// TIA Portal project "Digital – analógico (Ejercicio básico)" (V15.1)

(* hardware
DEVICE "S7-1200 station_2"  S7-1200 Station
   slot 0: "Rack_0"  S7-1200 Rack  Rack  V1.0
   slot 1: "PLC_2"  CPU 1214C AC/DC/Rly  6ES7 214-1BG40-0XB0  V4.1
   slot 3: "AQ 1x12BIT_1"  AQ1 signal board  6ES7 232-4HA30-0XB0  V1.0
*)

// ===== PLC "PLC_2"  CPU 1214C AC/DC/Rly =====

VAR_GLOBAL   // PLC tag table "Tabla de variables estándar"
   "etapa0" AT %M16.0 : Bool;
   "etapa1" AT %M16.1 : Bool;
   "etapa3" AT %M16.2 : Bool;
   "FC1" AT %I0.0 : Bool;
   "FC2" AT %I0.1 : Bool;
   "FC3" AT %I0.2 : Bool;
   "M" AT %I0.3 : Bool;
   "etapa2" AT %M16.3 : Bool;
   "Tag_1" AT %IW67 : Int;
   "Tag_2" AT %MD80 : Real;
   "Tag_3" AT %MD84 : Real;
   "Tag_4" AT %MD500 : DWord;
   "TAG9" AT %M500.0 : Bool;
   "Tag_5" AT %Q0.0 : Bool;
   "c100" AT %Q0.1 : Bool;
   "c10" AT %Q0.2 : Bool;
   "c-100" AT %Q0.3 : Bool;
   "Tag_6" AT %IW64 : Int;
   "Tag_7" AT %IW65 : Int;
   "Tag_8" AT %IW66 : Int;
   "Tag_9" AT %MD81 : DWord;
   "Tag_10" AT %MD82 : DWord;
   "Tag_11" AT %MD83 : DWord;
   "Tag_12" AT %IW80 : Word;
   "Tag_13" AT %IW81 : Word;
   "Tag_14" AT %MD30 : DWord;
   "Tag_15" AT %MD31 : DWord;
   "Tag_16" AT %MD32 : DWord;
   "Tag_17" AT %MD34 : Real;
   "Tag_18" AT %QW80 : Word;
END_VAR

FUNCTION "grafcet" : Void   // FC1, LAD
{ S7_Optimized_Access := 'TRUE' }
VERSION : 0.1
BEGIN

REGION Network 1
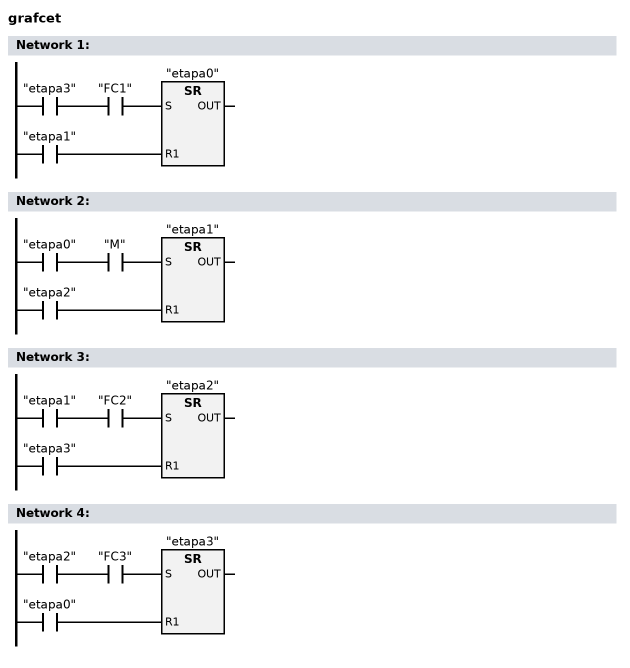
   RUNG wire#powerrail
      Contact( "etapa3" )
      Contact( "FC1" )
      S_SR(operand := "etapa0", r1 := wire#w1)
   END_RUNG
   RUNG wire#powerrail
      Contact( "etapa1" )
   END_RUNG wire#w1
   // the same network as SCL:
   IF "etapa3" AND "FC1" THEN
       "etapa0" := TRUE;   // SR flip-flop
   END_IF;
   IF "etapa1" THEN "etapa0" := FALSE; END_IF;
END_REGION

REGION Network 2
   RUNG wire#powerrail
      Contact( "etapa0" )
      Contact( "M" )
      S_SR(operand := "etapa1", r1 := wire#w1)
   END_RUNG
   RUNG wire#powerrail
      Contact( "etapa2" )
   END_RUNG wire#w1
   // the same network as SCL:
   IF "etapa0" AND "M" THEN
       "etapa1" := TRUE;   // SR flip-flop
   END_IF;
   IF "etapa2" THEN "etapa1" := FALSE; END_IF;
END_REGION

REGION Network 3
   RUNG wire#powerrail
      Contact( "etapa1" )
      Contact( "FC2" )
      S_SR(operand := "etapa2", r1 := wire#w1)
   END_RUNG
   RUNG wire#powerrail
      Contact( "etapa3" )
   END_RUNG wire#w1
   // the same network as SCL:
   IF "etapa1" AND "FC2" THEN
       "etapa2" := TRUE;   // SR flip-flop
   END_IF;
   IF "etapa3" THEN "etapa2" := FALSE; END_IF;
END_REGION

REGION Network 4
   RUNG wire#powerrail
      Contact( "etapa2" )
      Contact( "FC3" )
      S_SR(operand := "etapa3", r1 := wire#w1)
   END_RUNG
   RUNG wire#powerrail
      Contact( "etapa0" )
   END_RUNG wire#w1
   // the same network as SCL:
   IF "etapa2" AND "FC3" THEN
       "etapa3" := TRUE;   // SR flip-flop
   END_IF;
   IF "etapa0" THEN "etapa3" := FALSE; END_IF;
END_REGION
END_FUNCTION

FUNCTION "Irterak" : Void   // FC2, LAD
{ S7_Optimized_Access := 'TRUE' }
VERSION : 0.1
BEGIN

REGION Network 1
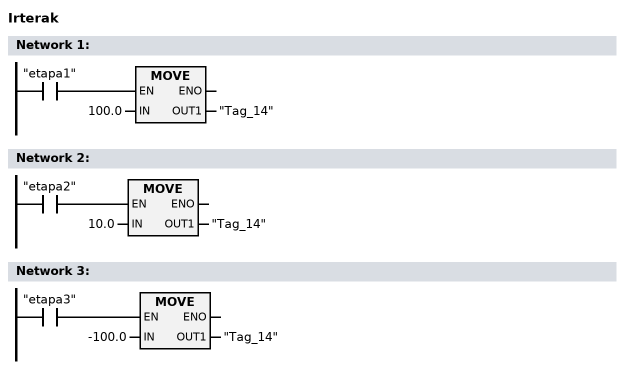
   RUNG wire#powerrail
      Contact( "etapa1" )
      Move(in := 100.0, out1 => "Tag_14")
   END_RUNG
   // the same network as SCL:
   IF "etapa1" THEN "Tag_14" := 100.0; END_IF;
END_REGION

REGION Network 2
   RUNG wire#powerrail
      Contact( "etapa2" )
      Move(in := 10.0, out1 => "Tag_14")
   END_RUNG
   // the same network as SCL:
   IF "etapa2" THEN "Tag_14" := 10.0; END_IF;
END_REGION

REGION Network 3
   RUNG wire#powerrail
      Contact( "etapa3" )
      Move(in := -100.0, out1 => "Tag_14")
   END_RUNG
   // the same network as SCL:
   IF "etapa3" THEN "Tag_14" := -100.0; END_IF;
END_REGION
END_FUNCTION

ORGANIZATION_BLOCK "Main"   // OB1, LAD, ProgramCycle
TITLE = "Main Program Sweep (Cycle)"
{ S7_Optimized_Access := 'TRUE' }
VERSION : 0.1
BEGIN

REGION Network 1
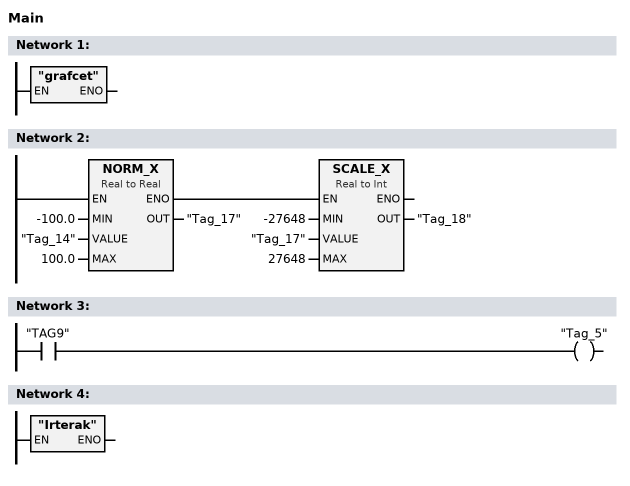
   RUNG wire#powerrail
      "grafcet"()
   END_RUNG
   // the same network as SCL:
   "grafcet"();
END_REGION

REGION Network 2
   RUNG wire#powerrail
      { S7_Templates := "[SrcType := Real, DestType := Real]"; S7_GenerateENO := "TRUE" } Normalize(min := -100.0, value := "Tag_14", max := 100.0, out => "Tag_17")
      { S7_Templates := "[SrcType := Real, DestType := Int]"; S7_GenerateENO := "TRUE" } Scale(min := -27648, value := "Tag_17", max := 27648, out => "Tag_18")
   END_RUNG
   // the same network as SCL:
   // ENO of a box is taken as its EN; it also drops when the box reports an error
   "Tag_17" := NORM_X(MIN := -100.0, VALUE := "Tag_14", MAX := 100.0);
   "Tag_18" := SCALE_X(MIN := -27648, VALUE := "Tag_17", MAX := 27648);
END_REGION

REGION Network 3
   RUNG wire#powerrail
      Contact( "TAG9" )
      Coil( "Tag_5" )
   END_RUNG
   // the same network as SCL:
   "Tag_5" := "TAG9";
END_REGION

REGION Network 4
   RUNG wire#powerrail
      "Irterak"()
   END_RUNG
   // the same network as SCL:
   "Irterak"();
END_REGION
END_ORGANIZATION_BLOCK

ORGANIZATION_BLOCK "Startup"   // OB100, LAD, Startup
TITLE = "Complete Restart"
{ S7_Optimized_Access := 'TRUE' }
VERSION : 0.1
   VAR_INPUT
      LostRetentive : Bool;   // True if retentive data are lost
      LostRTC : Bool;   // True if date and time are lost
   END_VAR
BEGIN

REGION Network 1
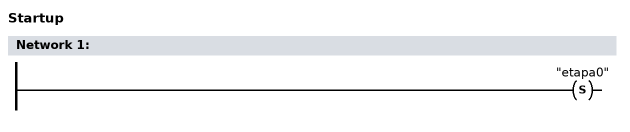
   RUNG wire#powerrail
      S_Coil( "etapa0" )
   END_RUNG
   // the same network as SCL:
   "etapa0" := TRUE;
END_REGION
END_ORGANIZATION_BLOCK